(* IEC 61131-3 sources: StewartPlatform/Class/SdiasManager (part 4) *)

END_FUNCTION

FUNCTION SdiasManager::DOL_Handling_Create_End_Cmd
	VAR_INPUT
		pEndCmdBuffer 	: ^t_SDIAS_DOListEntry;
	END_VAR

 	(* End of list	*)
	pEndCmdBuffer^.OffsetReadPayload := 0xFFFF;
	pEndCmdBuffer^.OffsetWritePayload := 0xFFFF;

	(* Set wait for DO to inactive	*)
	pEndCmdBuffer^.OffsetVolatileWaitFlag := SDIAS_INVALID_VOLATILE_WAIT_HANDLE;

	(* Init scratchpad info to 0	*)
	pEndCmdBuffer^.ErrorInfo := 0;

	pEndCmdBuffer^.CmdRetries := 0x0;

	pEndCmdBuffer^.ReadLength := 0;
	pEndCmdBuffer^.ReadOffset := 0;

	(* Init reserved info to 0	*)
	pEndCmdBuffer^.Reserved := 0;

	pEndCmdBuffer^.WriteLength := 0;
	pEndCmdBuffer^.WriteOffset  := 0;

END_FUNCTION

FUNCTION SdiasManager::LogSDOErrorInfo
	VAR_INPUT
		OSRetVal 	: DINT;
	END_VAR

 // show error info
  case OSRetVal of
    SDIAS_MAILBOX_FULL:
      LogValue("(SdiasManager::LogSDOErrorInfo) SDO Error 0x{0}: Mailbox full", (0-OSRetVal)$UDINT);

    SDIAS_TIMEOUT_TASK:
      LogValue("(SdiasManager::LogSDOErrorInfo) SDO Error 0x{0}: Timeout of task", (0-OSRetVal)$UDINT);

    SDIAS_RESPONSE_BUFFER_TOO_SMALL:
      LogValue("(SdiasManager::LogSDOErrorInfo) SDO Error 0x{0}: Response buffer too small", (0-OSRetVal)$UDINT);

    SDIAS_TIMEOUT_SDO_RESPONSE:
      LogValue("(SdiasManager::LogSDOErrorInfo) SDO Error 0x{0}: Timeout SDO response", (0-OSRetVal)$UDINT);

    SDIAS_OUT_OF_HANDLES:
      LogValue("(SdiasManager::LogSDOErrorInfo) SDO Error 0x{0}: Out of handles", (0-OSRetVal)$UDINT);

    SDIAS_INVALID_PARAM_DATA_LENGTH:
      LogValue("(SdiasManager::LogSDOErrorInfo) SDO Error 0x{0}: Invalid length of data bytes", (0-OSRetVal)$UDINT);

    SDIAS_INVALID_PARAM_DATA_BUFFER:
      LogValue("(SdiasManager::LogSDOErrorInfo) SDO Error 0x{0}: Invalid data buffer", (0-OSRetVal)$UDINT);

    SDIAS_INVALID_PARAM_SDO_HANDLE:
      LogValue("(SdiasManager::LogSDOErrorInfo) SDO Error 0x{0}: Invalid SDO handle", (0-OSRetVal)$UDINT);

    SDIAS_INVALID_PARAM_NODE:
      LogValue("(SdiasManager::LogSDOErrorInfo) SDO Error 0x{0}: Invalid node handle", (0-OSRetVal)$UDINT);

    SDIAS_GLOBAL_ERROR:
      LogValue("(SdiasManager::LogSDOErrorInfo) SDO Error 0x{0}: General Error of SDIAS Manager", (0-OSRetVal)$UDINT);

    SDIAS_INVALID_MANAGER:
      LogValue("(SdiasManager::LogSDOErrorInfo) SDO Error 0x{0}: SDIAS Manager not found", (0-OSRetVal)$UDINT);

    SDIAS_SENDING_SDO_REQUEST_FAILED:
      LogValue("(SdiasManager::LogSDOErrorInfo) SDO Error 0x{0}: Sending SDO request failed", (0-OSRetVal)$UDINT);

    SDIAS_RECEIVING_SDO_RESPONSE_FAILED:
      LogValue("(SdiasManager::LogSDOErrorInfo) SDO Error 0x{0}: Receiving SDO response failed", (0-OSRetVal)$UDINT);

    SDIAS_MANAGER_GLOBAL_ERROR:
      LogValue("(SdiasManager::LogSDOErrorInfo) SDO Error 0x{0}: General Error of SDIAS Manager (like communication problems to client)", (0-OSRetVal)$UDINT);

    SDIAS_INTERNAL_ERROR:
      LogValue("(SdiasManager::LogSDOErrorInfo) SDO Error 0x{0}: Internal error", (0-OSRetVal)$UDINT);
  else
    LogValue("(SdiasManager::LogSDOErrorInfo) SDO Error 0x{0}: Unknown Error", (0-OSRetVal)$UDINT);
  end_case;

END_FUNCTION

FUNCTION SdiasManager::CheckAccess
	VAR_INPUT
		bsStateByte 	: t_SDIAS_StateByte;
		sdRequired 	: DINT;
		sdPlace 	: DINT;
		pCrashThisTime 	: ^USINT;
		pCrashMessage 	: ^CHAR;
	END_VAR
	VAR_OUTPUT
		usRetryCounter 	: USINT;
	END_VAR

  // increase retrycounter if retries occured on the access
  usRetryCounter := bsStateByte SHR 5;

  // check if the access failed
  if sdRequired & (bsStateByte.AccessFailed = TRUE) then
    ModuleObjInfo[sdPlace].pThis^.ClassState := _RequiredError;
    RequiredPlace := sdPlace;
    CyclicMsgMarker.PostIt.RequiredError := TRUE;
    ClassState := _RequiredError;
    ErrorInitStep := InitSSW;
    InitSSW := _PrepareError;

    pCrashThisTime^ := 2;

    _strcpy(dest:=pCrashMessage, src:="Access to a required SDIAS Module failed");
  end_if;

END_FUNCTION

FUNCTION SdiasManager::PostRtMessages

  // if there are some messages to post, post them (the methods in the brackets are not the actual, but the methods were the error occured)
  if CyclicMsgMarker.PostIt then
    if CyclicMsgMarker.PostIt.IsoReadRunFailed then
      LogError("(SdiasManager::RtWork) Error changing the run state of the isochronous read access!");
    end_if;

    if CyclicMsgMarker.PostIt.IsoWriteRunFailed then
      LogError("(SdiasManager::RtWork) Error changing the run state of the isochronous write access!");
    end_if;

    if CyclicMsgMarker.PostIt.RequiredError then
      LogValue("(SdiasManager::RtWork) Required Error at SDIAS Place 0x{0}", RequiredPlace$UDINT);
    end_if;

    if CyclicMsgMarker.PostIt.ForwardRequiredErrorFailed then
      LogError("(SdiasManager::RtWork) Failed to set required error to BusInterface");
    end_if;

    if CyclicMsgMarker.PostIt.ToggleErrorWrTask & (CyclicMsgMarker.AlreadyPosted.ToggleErrorWrTask = FALSE) then
      LogError("(SdiasManager::RtWork) Error at toggle bit of iso write task of SDIAS");
      CyclicMsgMarker.AlreadyPosted.ToggleErrorWrTask := TRUE;
    end_if;

    if CyclicMsgMarker.PostIt.ToggleErrorRdTask & (CyclicMsgMarker.AlreadyPosted.ToggleErrorRdTask = FALSE) then
      LogError("(SdiasManager::RtWork) Error at toggle bit of iso read task of SDIAS");
      CyclicMsgMarker.AlreadyPosted.ToggleErrorRdTask := TRUE;
    end_if;

    if CyclicMsgMarker.PostIt.ErrorWrTask & (CyclicMsgMarker.AlreadyPosted.ErrorWrTask = FALSE) then
      LogValue("(SdiasManager::RtWork) Error at iso write task of SDIAS 0x{0}", (WriteTaskInfo.pReadData^.ErrorInfoFlags AND SDIAS_ERROR_INFO_MASK));
      CyclicMsgMarker.AlreadyPosted.ErrorWrTask := TRUE;
    end_if;

    if CyclicMsgMarker.PostIt.ErrorRdTask & (CyclicMsgMarker.AlreadyPosted.ErrorRdTask = FALSE) then
      LogValue("(SdiasManager::RtWork) Error at iso read task of SDIAS 0x{0}", (ReadTaskInfo.pReadData^.ErrorInfoFlags AND SDIAS_ERROR_INFO_MASK));
      CyclicMsgMarker.AlreadyPosted.ErrorRdTask := TRUE;
    end_if;

    if CyclicMsgMarker.PostIt.GetRdInfoFailed & (CyclicMsgMarker.AlreadyPosted.GetRdInfoFailed = FALSE) then
      LogError("(SdiasManager::RtWork) Error fetching iso read task info from OS");
      CyclicMsgMarker.AlreadyPosted.GetRdInfoFailed := TRUE;
    end_if;

    if CyclicMsgMarker.PostIt.GetWrInfoFailed & (CyclicMsgMarker.AlreadyPosted.GetWrInfoFailed = FALSE) then
      LogError("(SdiasManager::RtWork) Error fetching iso read task info from OS");
      CyclicMsgMarker.AlreadyPosted.GetWrInfoFailed := TRUE;
    end_if;

    if CyclicMsgMarker.PostIt.SetSyncFailed & (CyclicMsgMarker.AlreadyPosted.SetSyncFailed = FALSE) then
      LogError("(SdiasManager::RtWork) Failed to set sync out of pll");
      CyclicMsgMarker.AlreadyPosted.SetSyncFailed := TRUE;
    end_if;

    if CyclicMsgMarker.PostIt.GetFrameCounterFailed & (CyclicMsgMarker.AlreadyPosted.GetFrameCounterFailed = FALSE) then
      LogError("(SdiasManager::RtWork) Failed to get the frame counter info via OS interface");
      CyclicMsgMarker.AlreadyPosted.SetSyncFailed := TRUE;
    end_if;

    if CyclicMsgMarker.PostIt.WrTaskNotFinished & (CyclicMsgMarker.AlreadyPosted.WrTaskNotFinished = FALSE) then
      LogError("(SdiasManager::RtWork) Iso write task of SDIAS hasn't been completed");
      CyclicMsgMarker.AlreadyPosted.WrTaskNotFinished := TRUE;
    end_if;

    if CyclicMsgMarker.PostIt.WrTaskInterruptedByRdTask & (CyclicMsgMarker.AlreadyPosted.WrTaskInterruptedByRdTask = FALSE) then
      LogError("(SdiasManager::RtWork) Iso write task of SDIAS has been interrupted by read task");
      CyclicMsgMarker.AlreadyPosted.WrTaskInterruptedByRdTask := TRUE;
    end_if;

    if CyclicMsgMarker.PostIt.RdTaskNotFinished & (CyclicMsgMarker.AlreadyPosted.RdTaskNotFinished = FALSE) then
      // this happens on local SDIAS:
      //  - if the iso startpoint is too high and the SDIAS read task can't finish before the next RT
      //
      // on SDIAS via VARAN:
      //  - VARAN iso startpoint too low or SDIAS read task load too high => task is not finished when the data is fetched via VARAN
      LogError("(SdiasManager::RtWork) Iso read task of SDIAS hasn't been completed! Check setting of IsoStartPoint and cycle time!");
      CyclicMsgMarker.AlreadyPosted.RdTaskNotFinished := TRUE;
    end_if;
    if CyclicMsgMarker.PostIt.RdTaskNoEvent & (CyclicMsgMarker.AlreadyPosted.RdTaskNoEvent = FALSE) then
      // this happens on local SDIAS:
      //  - the RT takes too long and the SDIAS read task doesn't even start
      //
      // on SDIAS via VARAN:
      //  - VARAN iso startpoint or VARAN load too high => SDIAS read task doesn't even start
      LogError("(SdiasManager::RtWork) Iso read task of SDIAS hasn't been started! Check setting of IsoStartPoint and cycle time!");
      CyclicMsgMarker.AlreadyPosted.RdTaskNoEvent := TRUE;
    end_if;

    if CyclicMsgMarker.PostIt.TaskInfoRunFailed then
      LogError("(SdiasManager::RtWork) Error changing the run state of the isochronous read access to get the task info!");
    end_if;

    if CyclicMsgMarker.PostIt.IsoConfigWrTaskConfigFailed then
      LogError("(SdiasManager::RtWork) Error starting isochronous configuration write access with single for task config!");
    end_if;

    if CyclicMsgMarker.PostIt.IsoConfigWrTriggerUnitFailed then
      LogError("(SdiasManager::RtWork) Error starting isochronous configuration write access with single for trigger unit settings!");
    end_if;

    if CyclicMsgMarker.PostIt.IsoConfigWrChangeFailed then
      LogError("(SdiasManager::RtWork) Failed to change the isochronous configuration write access!");
    end_if;

    if CyclicMsgMarker.PostIt.IsoTaskConfigFailed then
      LogError("(SdiasManager::RtWork) Failed to set the iso read start config via OS interface!");
    end_if;

    if CyclicMsgMarker.PostIt.IsoTriggerUnitConfigFailed then
      LogError("(SdiasManager::RtWork) Failed to set the trigger unit config via OS interface!");
    end_if;

    if CyclicMsgMarker.PostIt.IsoConfigWrChange2Failed then
      LogError("(SdiasManager::RtWork) Error changing isochronous configuration write access for sync injection!");
    end_if;

    if CyclicMsgMarker.PostIt.IsoConfigWrSyncInjFailed then
      LogError("(SdiasManager::RtWork) Error starting isochronous configuration write access with single RUN for sync injection!");
    end_if;

    if CyclicMsgMarker.PostIt.IsoSyncInjFailed then
      LogError("(SdiasManager::RtWork) Failed to set the sync injection config via OS interface!");
    end_if;

    CyclicMsgMarker.PostIt := 0;
  end_if;

END_FUNCTION

FUNCTION SdiasManager::ChangeDynAccess
	VAR_INPUT
		AccessHandle 	: UDINT;
		NewOffset 	: HDINT;
		NewLength 	: UDINT;
	END_VAR
	VAR_OUTPUT
		Success 	: BOOL;
	END_VAR
  VAR
  	pAccess         : ^t_AccessElement;
    pControlStruct  : ^t_SDIAS_ControlStructDynamic;
  END_VAR

  Success := FALSE;

  // check if valid handle
  if AccessHandle then
    pAccess := AccessHandle$^t_AccessElement;

    if (pAccess^.eAccessType = _ReadDynamic) | (pAccess^.eAccessType = _WriteDynamic) then
      pControlStruct := (pAccess^.ppControlByte^)$^t_SDIAS_ControlStructDynamic;

      if pControlStruct then
        if NewOffset <> SDIAS_UNCHANGED_DYNAMIC_PARA then
          pControlStruct^.hiOffset := NewOffset$HINT + (pAccess^.usPlace shl 10);
        end_if;

        if NewLength <> SDIAS_UNCHANGED_DYNAMIC_PARA then
          pControlStruct^.usLength := NewLength$USINT;
        end_if;

        Success := TRUE;
      end_if;
    end_if;
  end_if;

END_FUNCTION

FUNCTION SdiasManager::CreateAndModifyIsoDOs
  VAR
    dataUPDATEDO          : t_UpdateDOCfg;
    dataADDDO             : t_AddDOCfg;
    dataResetDO           : t_ResetDOCfg;
  	tempCmd               : CmdStruct;
    _result               : results;
  END_VAR

  // initialize the data for the task config in realtime

  // set the task duration limit
  ISOTaskConfig.TaskDurationTimeout_us := (ud_BusTime_ns / 1000)$UINT;

  // start address of iso read list
  ISOTaskConfig.Config := gcMapping_Informations[IsoRdList].StartAddress;

  // we want to use the start configuration => enable it
  ISOTaskConfig.Config.SynchronizedStartEnable := TRUE;

  // initialize the data for the trigger unit setup for later use
  ISOTriggerUnitSetup.TaskSelect := 0;
  ISOTriggerUnitSetup.TaskSelect.IsoWrite := TRUE;
  ISOTriggerUnitSetup.TaskSelect.IsoRead  := TRUE;

  ISOTriggerUnitSetup.StartAddress := gcMapping_Informations[IsoWrPayload].StartAddress - SDIAS_TRIGGER_UNIT_BYTE_SIZE;
  ISOTriggerUnitSetup.StartAddress.UnitEnable := TRUE;

  if ConnectionType = SDIAS_CON_VIA_VARAN_uC then

    if b_IsoDOsCreated = FALSE then

#ifndef SDIAS_DEACTIVATE_TASK_CHECKS
      // DO for Task Infos (start at task 1 = read task)
      TaskInfoDO.Offset := SDIAS_OFFSET_TASK_INFO_1;
      TaskInfoDO.Length := sizeof(t_TaskInfoReadData);

      dataADDDO.Priority            := _BUS_IF_ISO_MOVE;
      dataADDDO.RdWr                := _BUS_IF_READ;
      dataADDDO.ud_addressoff_read  := TaskInfoDO.Offset;
      dataADDDO.ui_length_read      := TaskInfoDO.Length;
      dataADDDO.b_UseLocalCopy      := TRUE;

      tempCmd.uiCmd     := _BUS_IF_ADD_DO;
      tempCmd.aPara[0]  := (#dataADDDO)$DINT;

      ToBusInterface.NewInst(pPara:=#tempCmd, pResult:=#_result);
      if _result.aData[0]$t_BusIFRetvalErrorcode = _BUS_IF_RETVAL_OK then
        TaskInfoDO.Handle        := _result.aData$t_AddDORet.Handle;
        TaskInfoDO.pData         := _result.aData$t_AddDORet.pDataRead;
        TaskInfoDO.AccessHandle  := _result.aData$t_AddDORet.AccessHandle;

        // the parameter is overwritten with the DPRAM adress if the pData points to local memory
        TaskInfoDO.pDataDPRAM := dataADDDO.ud_addressoff_read$pVoid;
      else
        LogError("(SdiasManager::CreateAndModifyIsoDOs) Failed to add DO for the task info");
        InitError := _CreateDOFailed;
      end_if;
#endif

      // DO to enable read task in realtime before going to operational state
      dataADDDO.Priority            := _BUS_IF_ISO_MOVE;
      dataADDDO.RdWr                := _BUS_IF_WRITE;
      dataADDDO.ud_addressoff_write := SDIAS_OFFSET_TASK_CONFIG_1;
      dataADDDO.ui_length_write     := sizeof(t_TaskConfig);
      dataADDDO.b_UseLocalCopy      := TRUE;

      tempCmd.uiCmd     := _BUS_IF_ADD_DO;
      tempCmd.aPara[0]  := (#dataADDDO)$DINT;

      ToBusInterface.NewInst(pPara:=#tempCmd, pResult:=#_result);
      if _result.aData[0]$t_BusIFRetvalErrorcode = _BUS_IF_RETVAL_OK then
        ISOConfigWrDO.Handle        := _result.aData$t_AddDORet.Handle;
        ISOConfigWrDO.pData         := _result.aData$t_AddDORet.pDataWrite;
        ISOConfigWrDO.AccessHandle  := _result.aData$t_AddDORet.AccessHandle;

        // the parameter is overwritten with the DPRAM adress if the pData points to local memory
        ISOConfigWrDO.pDataDPRAM := dataADDDO.ud_addressoff_write$pVoid;

        // the first thing we write is the task config
        ISOConfigWrDO.pData^$t_TaskConfig := ISOTaskConfig;
      else
        LogError("(SdiasManager::CreateAndModifyIsoDOs) Failed to add DO for starting the iso read task");
        InitError := _CreateDOFailed;
      end_if;

      // recalculate payload size for accessing the payload

      // take our special access usage and add the usage according to the µC as well as 2 bytes for the trigger unit activation
      ISOWriteDO.Length += gcMapping_Informations[IsoWrPayload].ActUsage + SDIAS_TRIGGER_UNIT_BYTE_SIZE;

      // take our special access usage and add the usage according to the µC
      ISOReadDO.Length  += gcMapping_Informations[IsoRdPayload].ActUsage;

      // since we get the status info extra => skip the status byte of watchdog + status byte of write task info + write task info + status byte of read task info + read task info
      ISOReadDO.Length  -= sizeof(t_SDIAS_StateByte) + sizeof(t_SDIAS_StateByte) + sizeof(t_TaskInfoData.Handshake) + sizeof(t_TaskInfoData.DurationTime) + sizeof(t_TaskInfoData.ExecutionTime)
                                                     + sizeof(t_SDIAS_StateByte) + sizeof(t_TaskInfoData.Handshake) + sizeof(t_TaskInfoData.DurationTime) + sizeof(t_TaskInfoData.ExecutionTime);

      // Long DO for Read Data
      dataADDDO.Priority            := _BUS_IF_ISO_MOVE;
      dataADDDO.RdWr                := _BUS_IF_READ;
      dataADDDO.ud_addressoff_read  := 0;
      dataADDDO.ui_length_read      := ISOReadDO.Length;
      dataADDDO.b_UseLocalCopy      := TRUE;

      tempCmd.uiCmd     := _BUS_IF_ADD_DO;
      tempCmd.aPara[0]  := (#dataADDDO)$DINT;

      ToBusInterface.NewInst(pPara:=#tempCmd, pResult:=#_result);
      if _result.aData[0]$t_BusIFRetvalErrorcode = _BUS_IF_RETVAL_OK then
        ISOReadDO.Handle        := _result.aData$t_AddDORet.Handle;
        ISOReadDO.pData         := _result.aData$t_AddDORet.pDataRead;
        ISOReadDO.AccessHandle  := _result.aData$t_AddDORet.AccessHandle;

        // the parameter is overwritten with the DPRAM adress if the pData points to local memory
        ISOReadDO.pDataDPRAM := dataADDDO.ud_addressoff_read$pVoid;
      else
        LogError("(SdiasManager::CreateAndModifyIsoDOs) Failed to add long DO for the isochronous read data");
        InitError := _CreateDOFailed;
      end_if;

      // Long DO for Write Data
      dataADDDO.Priority            := _BUS_IF_ISO_MOVE;
      dataADDDO.RdWr                := _BUS_IF_WRITE;
      dataADDDO.ud_addressoff_write := 0;
      dataADDDO.ui_length_write     := ISOWriteDO.Length;
      dataADDDO.b_UseLocalCopy      := TRUE;

      tempCmd.uiCmd     := _BUS_IF_ADD_DO;
      tempCmd.aPara[0]  := (#dataADDDO)$DINT;

      ToBusInterface.NewInst(pPara:=#tempCmd, pResult:=#_result);
      if _result.aData[0]$t_BusIFRetvalErrorcode = _BUS_IF_RETVAL_OK then
        ISOWriteDO.Handle       := _result.aData$t_AddDORet.Handle;
        ISOWriteDO.pData        := _result.aData$t_AddDORet.pDataWrite;
        ISOWriteDO.AccessHandle := _result.aData$t_AddDORet.AccessHandle;

        // the parameter is overwritten with the DPRAM adress if the pData points to local memory
        ISOWriteDO.pDataDPRAM := dataADDDO.ud_addressoff_write$pVoid;
      else
        LogError("(SdiasManager::CreateAndModifyIsoDOs) Failed to add long DO for the isochronous write data");
        InitError := _CreateDOFailed;
      end_if;

      // reset data objects (calculate retry timeout)
      tempCmd.uiCmd     := _BUS_IF_RESET_DO;
      tempCmd.aPara[0]  := (#dataResetDO)$DINT;

      dataResetDO.Handle := ISOReadDO.Handle;

      ToBusInterface.NewInst(pPara:=#tempCmd, pResult:=#_result);
      if _result.aData[0]$t_BusIFRetvalErrorcode <> _BUS_IF_RETVAL_OK then
        LogError("(SdiasManager::CreateAndModifyIsoDOs) Failed reset long DO for the isochronous read data");
      end_if;

      dataResetDO.Handle := ISOWriteDO.Handle;

      ToBusInterface.NewInst(pPara:=#tempCmd, pResult:=#_result);
      if _result.aData[0]$t_BusIFRetvalErrorcode <> _BUS_IF_RETVAL_OK then
        LogError("(SdiasManager::CreateAndModifyIsoDOs) Failed reset long DO for the isochronous write data");
      end_if;

      if InitError <> _CreateDOFailed then
        b_IsoDOsCreated := TRUE;
        b_IsoDOsJustCreated := TRUE;
      end_if;
    end_if;
  end_if;

  // first we need to check out where our payload is stored and if it got the right size to access the right memory
  if gcMapping_Informations[IsoWrPayload].StartAddress then
    // modify if connected via VARAN
    if ConnectionType = SDIAS_CON_VIA_VARAN_uC then

                                                                                 // trigger unit is not actually part of the usage
      ISOWriteDO.Offset := gcMapping_Informations[IsoWrPayload].StartAddress - SDIAS_TRIGGER_UNIT_BYTE_SIZE; // the trigger unit starts earlier

      ISOWriteDO.pData^$UINT := ISOWriteDO.Length - SDIAS_TRIGGER_UNIT_BYTE_SIZE; // trigger unit itself is not part of the payload data size

      dataUPDATEDO.Handle               := ISOWriteDO.Handle;
      dataUPDATEDO.ud_addressoff_write  := ISOWriteDO.Offset;
      dataUPDATEDO.ud_length_write      := ISOWriteDO.Length;

      tempCmd.uiCmd         := _BUS_IF_UPDATE_DO;
      tempCmd.aPara[0]      := (#dataUPDATEDO)$DINT;

      ToBusInterface.NewInst(pPara:=#tempCmd, pResult:=#_result);
      if _result.aData[0]$t_BusIFRetvalErrorcode <> _BUS_IF_RETVAL_OK then
        LogError("(SdiasManager::CreateAndModifyIsoDOs) Failed to change isochronous write access! Unable to continue with Initialisation!");
        ClassState := _ManagerError;
        ErrorInitStep := InitSSW;
        InitSSW := _PrepareError;
        return;
      end_if;
    else
      // create if connected locally

      // Long DO for Write Data

      // take our special access usage and add the usage according to the µC as well as 2 bytes for the trigger unit activation
      ISOWriteDO.Length += gcMapping_Informations[IsoWrPayload].ActUsage + SDIAS_TRIGGER_UNIT_BYTE_SIZE;

      ISOWriteDO.Offset := gcMapping_Informations[IsoWrPayload].StartAddress - SDIAS_TRIGGER_UNIT_BYTE_SIZE; // the trigger unit starts earlier

      dataADDDO.Priority            := _BUS_IF_ISO_MOVE;
      dataADDDO.RdWr                := _BUS_IF_WRITE;
      dataADDDO.ud_addressoff_write := ISOWriteDO.Offset;
      dataADDDO.ui_length_write     := ISOWriteDO.Length;
      dataADDDO.ud_addressoff_read  := 0;
      dataADDDO.ui_length_read      := 0;
      dataADDDO.b_UseLocalCopy      := TRUE;

      tempCmd.uiCmd     := _BUS_IF_ADD_DO;
      tempCmd.aPara[0]  := (#dataADDDO)$DINT;

      ToBusInterface.NewInst(pPara:=#tempCmd, pResult:=#_result);
      if _result.aData[0]$t_BusIFRetvalErrorcode = _BUS_IF_RETVAL_OK then
        ISOWriteDO.Handle       := _result.aData$t_AddDORet.Handle;
        ISOWriteDO.pData        := _result.aData$t_AddDORet.pDataWrite;
        ISOWriteDO.AccessHandle := _result.aData$t_AddDORet.AccessHandle;

        // initialize the trigger unit
        ISOWriteDO.pData^$UINT := ISOWriteDO.Length - SDIAS_TRIGGER_UNIT_BYTE_SIZE;

        // the parameter is overwritten with the DPRAM adress if the pData points to local memory
        ISOWriteDO.pDataDPRAM := dataADDDO.ud_addressoff_write$pVoid;
      else
        LogError("(SdiasManager::CreateAndModifyIsoDOs) Failed to add long DO for the isochronous write data");
        InitError := _CreateDOFailed;
      end_if;
    end_if;
  end_if;

  if gcMapping_Informations[IsoRdPayload].StartAddress then
    // modify if connected via VARAN
    if ConnectionType = SDIAS_CON_VIA_VARAN_uC then
      ISOReadDO.Offset := gcMapping_Informations[IsoRdPayload].StartAddress;

      // since we get the status info extra => skip the status byte of watchdog + status byte of write task info + write task info + status byte of read task info + read task info
      ISOReadDO.Offset += sizeof(t_SDIAS_StateByte) + sizeof(t_SDIAS_StateByte) + sizeof(t_TaskInfoData.Handshake) + sizeof(t_TaskInfoData.DurationTime) + sizeof(t_TaskInfoData.ExecutionTime)
                                                    + sizeof(t_SDIAS_StateByte) + sizeof(t_TaskInfoData.Handshake) + sizeof(t_TaskInfoData.DurationTime) + sizeof(t_TaskInfoData.ExecutionTime);

      dataUPDATEDO.Handle               := ISOReadDO.Handle;
      dataUPDATEDO.ud_addressoff_read   := ISOReadDO.Offset;
      dataUPDATEDO.ud_length_read       := ISOReadDO.Length;

      tempCmd.uiCmd         := _BUS_IF_UPDATE_DO;
      tempCmd.aPara[0]      := (#dataUPDATEDO)$DINT;

      ToBusInterface.NewInst(pPara:=#tempCmd, pResult:=#_result);
      if _result.aData[0]$t_BusIFRetvalErrorcode <> _BUS_IF_RETVAL_OK then
        LogError("(SdiasManager::CreateAndModifyIsoDOs) Failed to change isochronous read access! Unable to continue with Initialisation!");
        ClassState := _ManagerError;
        ErrorInitStep := InitSSW;
        InitSSW := _PrepareError;
        return;
      end_if;
    else
      // create if connected locally

      // Long DO for Read Data

      // take our special access usage and add the usage according to the µC
      ISOReadDO.Length  += gcMapping_Informations[IsoRdPayload].ActUsage;

      ISOReadDO.Offset := gcMapping_Informations[IsoRdPayload].StartAddress;

      dataADDDO.Priority            := _BUS_IF_ISO_MOVE;
      dataADDDO.RdWr                := _BUS_IF_READ;
      dataADDDO.ud_addressoff_read  := ISOReadDO.Offset;
      dataADDDO.ui_length_read      := ISOReadDO.Length;
      dataADDDO.ud_addressoff_write := 0;
      dataADDDO.ui_length_write     := 0;
      dataADDDO.b_UseLocalCopy      := TRUE;

      tempCmd.uiCmd     := _BUS_IF_ADD_DO;
      tempCmd.aPara[0]  := (#dataADDDO)$DINT;

      ToBusInterface.NewInst(pPara:=#tempCmd, pResult:=#_result);
      if _result.aData[0]$t_BusIFRetvalErrorcode = _BUS_IF_RETVAL_OK then
        ISOReadDO.Handle        := _result.aData$t_AddDORet.Handle;
        ISOReadDO.pData         := _result.aData$t_AddDORet.pDataRead;
        ISOReadDO.AccessHandle  := _result.aData$t_AddDORet.AccessHandle;

        // the parameter is overwritten with the DPRAM adress if the pData points to local memory
        ISOReadDO.pDataDPRAM := dataADDDO.ud_addressoff_read$pVoid;
      else
        LogError("(SdiasManager::CreateAndModifyIsoDOs) Failed to add long DO for the isochronous read data");
        InitError := _CreateDOFailed;
      end_if;
    end_if;
  end_if;

END_FUNCTION

FUNCTION SdiasManager::IsDeviceBitSet
	VAR_INPUT
		pDeviceBitMap 	: ^BDINT;
		Place 	: UDINT;
	END_VAR
	VAR_OUTPUT
		bIsSet 	: BOOL;
	END_VAR

  if Place >= 32 then
    Place -= 32;
    pDeviceBitmap += 4;
  end_if;
  bIsSet := ((pDeviceBitmap^ SHR Place) AND 1)$BOOL;

END_FUNCTION

FUNCTION SdiasManager::DisableBus
  VAR
    dataSETRUNSTATE     : t_SetRunStateCfg;
  	tempCmd             : CmdStruct;
    _result             : results;
    dataUPDATEDO        : t_UpdateDOCfg;
    aProperties         : ARRAY [0..4] OF SDM_PROPERTY_VALUE_PAIR;
    SyncInjectionCfg    : t_SyncInjectionCfg;
  END_VAR

  // we select the read task for sync, there are no sync task trigger losses allowed and we disable the sync injection
  SyncInjectionCfg := 16#02;

  if ConnectionType = SDIAS_CON_VIA_VARAN_uC then
    // change config DO => change trigger unit settings (also use trigger unit for read task)
    ISOConfigWrDO.Offset := SDIAS_OFFSET_SYNC_INJECTION_CFG;
    ISOConfigWrDO.Length := sizeof(t_SyncInjectionCfg);

    dataUPDATEDO.Handle               := ISOConfigWrDO.Handle;
    dataUPDATEDO.ud_addressoff_write  := ISOConfigWrDO.Offset;
    dataUPDATEDO.ud_length_write      := ISOConfigWrDO.Length;

    tempCmd.uiCmd         := _BUS_IF_UPDATE_DO;
    tempCmd.aPara[0]      := (#dataUPDATEDO)$DINT;

    ToBusInterface.NewInst(pPara:=#tempCmd, pResult:=#_result);

    if _result.aData[0]$t_BusIFRetvalErrorcode <> _BUS_IF_RETVAL_OK then
      // remember the log message and write it in cyclic priority to avoid a rt runtime error
      CyclicMsgMarker.PostIt.IsoConfigWrChange2Failed := TRUE;
    else
      // use the sync injection data
      ISOConfigWrDO.pData^$t_SyncInjectionCfg := SyncInjectionCfg;
    end_if;

    dataSETRUNSTATE.NewRunState := _BUS_IF_RUN_STATE_SINGLE_RUN;
    tempCmd.uiCmd               := _BUS_IF_SET_RUN_STATE;
    tempCmd.aPara[0]            := (#dataSETRUNSTATE)$DINT;

    dataSETRUNSTATE.Handle      := ISOConfigWrDO.Handle;

    ToBusInterface.NewInst(pPara:=#tempCmd, pResult:=#_result);

    if _result.aData[0]$t_BusIFRetvalErrorcode <> _BUS_IF_RETVAL_OK then
      // remember the log message and write it in cyclic priority to avoid a rt runtime error
      CyclicMsgMarker.PostIt.IsoConfigWrSyncInjFailed := TRUE;
    end_if;
  else
    aProperties[0].udPropertyId     := SDM_PROP_SYNC_INJECTION_CONFIG;
    aProperties[0].udPropertyValue  := SyncInjectionCfg;

    if SDIAS_iSetNodeProperties(hNodeHandle         := udNodeHandle
                              , udPropertyCount     := 1
                              , psPropertyValuePairs:= #aProperties[0]
                              ) <> SDIAS_OK then
      // remember the log message and write it in cyclic priority to avoid a rt runtime error
      CyclicMsgMarker.PostIt.IsoSyncInjFailed := TRUE;
    end_if;
  end_if;

  // general settings needed for all DOs
  dataSETRUNSTATE.NewRunState := _BUS_IF_RUN_STATE_NO_RUN;
  tempCmd.uiCmd         := _BUS_IF_SET_RUN_STATE;
  tempCmd.aPara[0]      := (#dataSETRUNSTATE)$DINT;

#ifndef SDIAS_DEACTIVATE_TASK_CHECKS
  if ConnectionType = SDIAS_CON_VIA_VARAN_uC then
    // set runstate of taskinfo read
    dataSETRUNSTATE.Handle      := TaskInfoDO.Handle;

    ToBusInterface.NewInst(pPara:=#tempCmd, pResult:=#_result);

    if _result.aData[0]$t_BusIFRetvalErrorcode <> _BUS_IF_RETVAL_OK then
      // remember the log message and write it in cyclic priority to avoid a rt runtime error
      CyclicMsgMarker.PostIt.TaskInfoRunFailed := TRUE;
    end_if;
  end_if;
#endif

  // set runstate of read
  dataSETRUNSTATE.Handle      := ISOReadDO.Handle;

  ToBusInterface.NewInst(pPara:=#tempCmd, pResult:=#_result);

  if _result.aData[0]$t_BusIFRetvalErrorcode <> _BUS_IF_RETVAL_OK then
    // remember the log message and write it in cyclic priority to avoid a rt runtime error
    CyclicMsgMarker.PostIt.IsoReadRunFailed := TRUE;
  end_if;

  // set runstate of write
  dataSETRUNSTATE.Handle      := ISOWriteDO.Handle;

  ToBusInterface.NewInst(pPara:=#tempCmd, pResult:=#_result);

  if _result.aData[0]$t_BusIFRetvalErrorcode <> _BUS_IF_RETVAL_OK then
    // remember the log message and write it in cyclic priority to avoid a rt runtime error
    CyclicMsgMarker.PostIt.IsoWriteRunFailed := TRUE;
  end_if;

END_FUNCTION

FUNCTION GLOBAL SdiasManager::BusIFLogIn
  VAR
  	tempCmd         : CmdStruct;
    _result         : results;
    dataADDCallback : t_BusIFAddCallback;
  END_VAR

  // first check if the module may be deactivated
  tempCmd.uiCmd     := _BUS_IF_GET_DEACTIVATED_STATE;
  ToBusInterface.NewInst(pPara:=#tempCmd, pResult:=#_result);
  if _result.aData[0]$t_BusIFRetvalErrorcode = _BUS_IF_RETVAL_OK then
    b_Deactivated := _result.aData[4]$BOOL;
    if b_Deactivated then
      LogError("(SdiasManager::BusIFLogIn) SDIAS Manager object inactive");
      return;
    end_if;
  else
    LogError("(SdiasManager::BusIFLogIn) Failed to get deactivation state via BusInterface");
  end_if;

  // Set this class as the operator class of the BusInterface
  dataADDCallback.pthis := this$pVirtualBase;

  tempCmd.uiCmd     := _BUS_IF_ADD_CALLBACK;
  tempCmd.aPara[0]  := (#dataADDCallback)$DINT;
  ToBusInterface.NewInst(pPara:=#tempCmd, pResult:=#_result);
  if _result.aData[0]$t_BusIFRetvalErrorcode <> _BUS_IF_RETVAL_OK then
    LogError("(SdiasManager::BusIFLogIn) Failed to install callback at bus interface");
  else
    b_CallbackAdded := TRUE;
  end_if;

END_FUNCTION

FUNCTION SdiasManager::SendPostInitFinished
	VAR_INPUT
		DisableThisObject 	: BOOL;(* := FALSE *)
	END_VAR
  VAR
  	tempCmd         : CmdStruct;
    _result         : results;
  END_VAR

  b_PostInitFinished := TRUE;
  tempCmd.uiCmd := _BUS_IF_POST_INIT_FINISHED;
  ToBusInterface.NewInst(pPara:=#tempCmd, pResult:=#_result);

  if _result.aData[0]$t_BusIFRetvalErrorcode <> _BUS_IF_RETVAL_OK then
    LogError("(SdiasManager::CyWork) Failed to set the post init to finished via bus interface!");
  end_if;

  if DisableThisObject then
    // tell the manager that we don't need to be called for rt syncing
    tempCmd.uiCmd := _BUS_IF_RT_SYNC_READY;
    ToBusInterface.NewInst(pPara:=#tempCmd, pResult:=#_result);

    if _result.aData[0]$t_BusIFRetvalErrorcode <> _BUS_IF_RETVAL_OK then
      LogError("(SdiasManager::CyWork) Failed to set rt sync ready via bus interface!");
    end_if;
  end_if;

END_FUNCTION
